(* CoDeSys 2.3.9.41 project: Tutorial.pro *)
(* Libraries: Util.lib*18.5.10 15:14:28, ÏËÊ_Ï×Â_v2.lib 26.7.19 14:18:06, STANDARD.LIB 4.10.05 11:14:46, IECSFC.LIB 13.4.06 15:51:28, SYSLIBTIME.LIB 20.2.06 12:31:16, SYSTASKINFO.LIB 20.2.06 12:31:38, ANALYZATION.LIB 5.10.99 09:05:06, SYSLIBCALLBACK.LIB 20.2.06 12:31:08 *)

(* PLC configuration (modules and I/O channels)
Discrete input 8 bit [ID100] node 0, in %IB0 out %QB0 {Filtrationtime = 10; Filtrationtime = 10; Filtrationtime = 10; Filtrationtime = 10; Filtrationtime = 10; Filtrationtime = 10; Filtrationtime = 10; Filtrationtime = 10; Visibility = No; PinCount = 8; WatchDogPeriod = 1000; PollPeriod = 1}
  AT %IB0.0 [ByteInput] 8 discrete inputs
Discrete output 2 bit [ID101] node 1, in %IB1 out %QB1 {PinCount = 2; SafeValueBool = FALSE; SafeValueBool = FALSE; Visibility = No}
  AT %QX1.0 [BitOutput] First
  AT %QX1.1 [BitOutput] Second
Discrete output 2 bit [ID101] node 2, in %IB2 out %QB2 {PinCount = 2; SafeValueBool = FALSE; SafeValueBool = FALSE; Visibility = No}
  AT %QX2.0 [BitOutput] First
  AT %QX2.1 [BitOutput] Second
Discrete output 2 bit [ID101] node 3, in %IB3 out %QB3 {PinCount = 2; SafeValueBool = FALSE; SafeValueBool = FALSE; Visibility = No}
  AT %QX3.0 [BitOutput] First
  AT %QX3.1 [BitOutput] Second
Discrete output 2 bit [ID101] node 4, in %IB4 out %QB4 {PinCount = 2; SafeValueBool = FALSE; SafeValueBool = FALSE; Visibility = No}
  AT %QX4.0 [BitOutput] First
  AT %QX4.1 [BitOutput] Second
Discrete output 2 bit [ID101] node 5, in %IB5 out %QB5 {PinCount = 2; SafeValueBool = FALSE; SafeValueBool = FALSE; Visibility = No}
  AT %QX5.0 [BitOutput] First
  AT %QX5.1 [BitOutput] Second
Discrete output 2 bit [ID101] node 6, in %IB6 out %QB6 {PinCount = 2; SafeValueBool = FALSE; SafeValueBool = FALSE; Visibility = No}
  AT %QX6.0 [BitOutput] First
  AT %QX6.1 [BitOutput] Second
Special output [ID104] node 7, in %IB7 out %QB7 {Visibility = No; PinCount = 1}
  AT %QX7.0 [BitOutput] Special output
AT %QD8.0 [DWordOutput] Last address
AT %QW8.1 [WordOutput] Last error
RS-485-1 [COM1_USART] node 0, in %IB8.0 out %QB8.0 {CommunicationSpeed = 9600; Parity = NO PARITY CHECK; BitLength = 8 bits; StopLength = One stop bit; InterfaceType = RS485; FrameOriented = RTU; Timeout = 0; Visibility = No}
AT %QB8.1.0 [ComChannel] Command (0xff - Start)
Register output module [ID2004] node 0, in %IB8.1.0 out %QB8.1.0 {ModbusAddress = 49999; Command_write_one_reg = Write multiple registers(0x10); Visibility = No}
  comWord AT %QW8.1.0.0 [WordOutput]
Register input module [ID2003] node 1, in %IB8.1.1 out %QB8.1.1 {ModbusAddress = 50199; Command_read_regs = Read holding Registers  (0x03); Visibility = No}
  statusWord AT %IW8.1.1.0 [WordInput]
Register output module [ID2004] node 2, in %IB8.1.2 out %QB8.1.2 {ModbusAddress = 50009; Command_write_one_reg = Write multiple registers(0x10); Visibility = No}
  tsk AT %QW8.1.2.0 [WordOutput]
32bit output module [ID2006] node 3, in %IB8.1.3 out %QB8.1.3 {ModbusAddress = 3019; Command_write_regs = Preset multiple Registers (0x10); Visibility = No}
  tsk_min AT %QD8.1.3.0 [DWordOutput]
32bit output module [ID2006] node 4, in %IB8.1.4 out %QB8.1.4 {ModbusAddress = 3029; Command_write_regs = Preset multiple Registers (0x10); Visibility = No}
  tsk_max AT %QD8.1.4.0 [DWordOutput]
Register output module [ID2004] node 5, in %IB8.1.5 out %QB8.1.5 {ModbusAddress = 3099; Command_write_one_reg = Write multiple registers(0x10); Visibility = No}
  pre_tsk AT %QW8.1.5.0 [WordOutput]
Register output module [ID2004] node 6, in %IB8.1.6 out %QB8.1.6 {ModbusAddress = 8; Command_write_one_reg = Write multiple registers(0x10); Visibility = No}
  p_t_num AT %QW8.1.6.0 [WordOutput]
Register output module [ID2004] node 7, in %IB8.1.7 out %QB8.1.7 {ModbusAddress = 4139; Command_write_one_reg = Write multiple registers(0x10); Visibility = No}
  lim AT %QW8.1.7.0 [WordOutput]
Register output module [ID2004] node 8, in %IB8.1.8 out %QB8.1.8 {ModbusAddress = 2009; Command_write_one_reg = Write multiple registers(0x10); Visibility = No}
  idc_st AT %QW8.1.8.0 [WordOutput]
Register output module [ID2004] node 9, in %IB8.1.9 out %QB8.1.9 {ModbusAddress = 3149; Command_write_one_reg = Write multiple registers(0x10); Visibility = No}
  rs_ AT %QW8.1.9.0 [WordOutput]
Register input module [ID2003] node 10, in %IB8.1.10 out %QB8.1.10 {ModbusAddress = 16099; Command_read_regs = Read holding Registers  (0x03); Visibility = No}
  p_val AT %IW8.1.10.0 [WordInput]
Register input module [ID2003] node 11, in %IB8.1.11 out %QB8.1.11 {ModbusAddress = 16119; Command_read_regs = Read holding Registers  (0x03); Visibility = No}
  U_val AT %IW8.1.11.0 [WordInput]
  f_val AT %IW8.1.12.0 [WordInput]
  i_val AT %IW8.1.13.0 [WordInput]
*)

(* POU PLC_PRG, CFC *)
PROGRAM PLC_PRG
VAR
	n1:BYTE:=1;
	st1:BOOL;
	st2:BOOL;
	st3:BOOL;
	s1:BOOL:=TRUE;
	r1:BOOL;
	com1: com_word_fb;
	statFB: stat_word_fb;
	taskfb: task_fb;
	r_eng: BOOL;
	r_drv: BOOL;
	sl_st: BOOL;
	al: BOOL;
	war: BOOL;
	tsk_st: BOOL;
	r_a: BOOL;
	range: BOOL;
	w_st: BOOL;
	v_st: BOOL;
	cur_st: BOOL;
	heat_st: BOOL;
	Pn: REAL;
	Un: REAL;
	fn: REAL;
	In: REAL;
	tmin1: REAL;
	tmax1: REAL:=50;
	tsk1: REAL:=30;
	p_tsk1: REAL;
	p_tsk2: REAL;
	p_tsk3: REAL;
	p_tsk4: REAL;
	lim_high1: REAL:=50;
	Idc_s1: WORD:=10;
	r_off: BOOL;
	valuefb: value_fb;
END_VAR
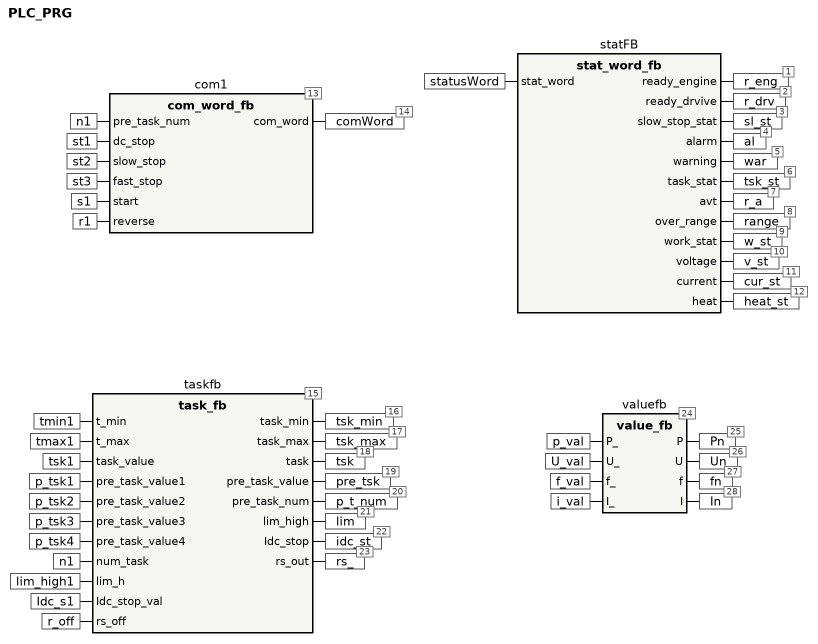
_CFC_ (* Continuous Function Chart, elements in execution order *)
#0 statFB:stat_word_fb(stat_word: statusWord)
#1 r_eng <= #0.ready_engine
#2 r_drv <= #0.ready_drvive
#3 sl_st <= #0.slow_stop_stat
#4 al <= #0.alarm
#5 war <= #0.warning
#6 tsk_st <= #0.task_stat
#7 r_a <= #0.avt
#8 range <= #0.over_range
#9 w_st <= #0.work_stat
#10 v_st <= #0.voltage
#11 cur_st <= #0.current
#12 heat_st <= #0.heat
#13 com1:com_word_fb(pre_task_num: n1, dc_stop: st1, slow_stop: st2, fast_stop: st3, start: s1, reverse: r1)
#14 comWord <= #13.com_word
#15 taskfb:task_fb(t_min: tmin1, t_max: tmax1, task_value: tsk1, pre_task_value1: p_tsk1, pre_task_value2: p_tsk2, pre_task_value3: p_tsk3, pre_task_value4: p_tsk4, num_task: n1, lim_h: lim_high1, Idc_stop_val: Idc_s1, rs_off: r_off)
#16 tsk_min <= #15.task_min
#17 tsk_max <= #15.task_max
#18 tsk <= #15.task
#19 pre_tsk <= #15.pre_task_value
#20 p_t_num <= #15.pre_task_num
#21 lim <= #15.lim_high
#22 idc_st <= #15.Idc_stop
#23 rs_ <= #15.rs_out
#24 valuefb:value_fb(P_: p_val, U_: U_val, f_: f_val, I_: i_val)
#25 Pn <= #24.P
#26 Un <= #24.U
#27 fn <= #24.f
#28 In <= #24.I
_END_CFC_
(* the same logic as Structured Text *)
statFB(stat_word := statusWord);
r_eng := statFB.ready_engine;
r_drv := statFB.ready_drvive;
sl_st := statFB.slow_stop_stat;
al := statFB.alarm;
war := statFB.warning;
tsk_st := statFB.task_stat;
r_a := statFB.avt;
range := statFB.over_range;
w_st := statFB.work_stat;
v_st := statFB.voltage;
cur_st := statFB.current;
heat_st := statFB.heat;
com1(pre_task_num := n1, dc_stop := st1, slow_stop := st2, fast_stop := st3, start := s1, reverse := r1);
comWord := com1.com_word;
taskfb(t_min := tmin1, t_max := tmax1, task_value := tsk1, pre_task_value1 := p_tsk1, pre_task_value2 := p_tsk2, pre_task_value3 := p_tsk3, pre_task_value4 := p_tsk4, num_task := n1, lim_h := lim_high1, Idc_stop_val := Idc_s1, rs_off := r_off);
tsk_min := taskfb.task_min;
tsk_max := taskfb.task_max;
tsk := taskfb.task;
pre_tsk := taskfb.pre_task_value;
p_t_num := taskfb.pre_task_num;
lim := taskfb.lim_high;
idc_st := taskfb.Idc_stop;
rs_ := taskfb.rs_out;
valuefb(P_ := p_val, U_ := U_val, f_ := f_val, I_ := i_val);
Pn := valuefb.P;
Un := valuefb.U;
fn := valuefb.f;
In := valuefb.I;
END_PROGRAM
